TYPE ST_ACStatus :
STRUCT
	OnOff: BOOL;
	mode: INT;
	HorizSwingOnOff: BOOL;
	VertiSwingOnOff: BOOL;
	temp: REAL;
END_STRUCT
END_TYPE

(* stored: Version 1.1.0.1, ProductVersion 3.1.4024.12
   DUT ST_ACStatus: Id {d4780a66-bdb0-426c-8252-88435ec565c6} *)
